FUNCTION AdsLogMessage : BOOL
VAR_INPUT
  sMessage : STRING;
END_VAR
VAR
  sMsgFormat : STRING := 'PLC Msg: %s';
  msgCtrlMask : DWORD := ADSLOG_MSGTYPE_HINT OR ADSLOG_MSGTYPE_LOG;
END_VAR


ADSLOGSTR(msgCtrlMask:= msgCtrlMask, msgFmtStr:= sMsgFormat, strArg:= sMessage);

END_FUNCTION

(* stored: Version 1.1.0.1, ProductVersion 3.1.4024.12
   POU AdsLogMessage: Id {01c57617-6b09-4dca-b186-b80054f005eb}, SpecialFunc None *)
